(* CoDeSys 2.3 export: GETEEP_PAGE.EXP *)

(* POU 05_Basic_Calc/eeprom_operations/getEEP_Page, ST *)
(* Определение номера страницы eeprom по индексу параметра *)
FUNCTION getEEP_Page : INT
VAR_INPUT
	EEP_num					: INT;
END_VAR
VAR
	EEP_ELEMENT_OF_PAGE	: INT		:= 256;
END_VAR
getEEP_Page := EEP_num / EEP_ELEMENT_OF_PAGE;
END_FUNCTION
